{attribute addProperty BoxType "EL6201-0000-0017"}
{attribute addProperty Id "Slave_10A_DO0BIT10.12573Slave_10A_DO1BIT10.12574Slave_10A_DO2BIT10.12575Slave_10A_DO3BIT10.12576Slave_10B_DO0BIT10.12577Slave_10B_DO1BIT10.12578Slave_10B_DO2BIT10.12579Slave_10B_DO3BIT10.12580"}
{attribute addProperty CRC "3166583453"}
{attribute addProperty SizeInBites "8"}
{attribute addProperty SizeInBytes "1"}
TYPE Slave_10_Outputs_BCBE3A9D :
STRUCT
	{attribute addProperty Name "Slave_10A_DO0"}
	Slave_10A_DO0 : BIT;
	{attribute addProperty Name "Slave_10A_DO1"}
	Slave_10A_DO1 : BIT;
	{attribute addProperty Name "Slave_10A_DO2"}
	Slave_10A_DO2 : BIT;
	{attribute addProperty Name "Slave_10A_DO3"}
	Slave_10A_DO3 : BIT;
	{attribute addProperty Name "Slave_10B_DO0"}
	Slave_10B_DO0 : BIT;
	{attribute addProperty Name "Slave_10B_DO1"}
	Slave_10B_DO1 : BIT;
	{attribute addProperty Name "Slave_10B_DO2"}
	Slave_10B_DO2 : BIT;
	{attribute addProperty Name "Slave_10B_DO3"}
	Slave_10B_DO3 : BIT;
END_STRUCT
END_TYPE

(* stored: Version 1.2.0.0, ProductVersion 3.1.4024.9
   DUT Slave_10_Outputs_BCBE3A9D: Id {23bbb8c9-31bc-4c2f-87bc-9f6cffc409de} *)
